(* CoDeSys 2.3 export: FB_SYNC_JALOUSIE_DELAY.EXP *)

(* POU FBs/FB_SYNC_JALOUSIE_DELAY, ST *)
FUNCTION_BLOCK FB_SYNC_JALOUSIE_DELAY
VAR_INPUT
	IN: BOOL;
	nextZeroVoltage: T_DCTIME;
END_VAR
VAR_OUTPUT
	Q AT %Q*: BOOL;
END_VAR
VAR
	fbDrand: DRAND;
END_VAR
Q := IN;
END_FUNCTION_BLOCK
